KUKA KRL program: init_real.src

&ACCESS RVO1
&COMMENT
DEFFCT REAL init_real(r :IN, rDefault :IN)
INT r, rDefault

IF Varstate("r") <> #initialized THEN
  IF Varstate("rDefault") <> #initialized THEN
    RETURN 0.0
  ENDIF
  RETURN rDefault
ENDIF

RETURN r

ENDFCT
